{attribute 'GeneratedUsingTerminal: AMP8000-0030-0103-0103'}
{attribute addProperty BoxType "AMP8000-0030-0103-0103"}
{attribute addProperty Id "WcState0AT %I*BOOL1WcState1AT %I*BOOL1InputToggle0AT %I*BOOL1InputToggle1AT %I*BOOL1"}
{attribute addProperty CRC "3038159460"}
{attribute addProperty Size "4"}
TYPE WcState_B516A264 :
STRUCT
	{attribute addProperty Name "WcState0"}
	WcState0 AT %I* : BOOL;
	{attribute addProperty Name "WcState1"}
	WcState1 AT %I* : BOOL;
	{attribute addProperty Name "InputToggle0"}
	InputToggle0 AT %I* : BOOL;
	{attribute addProperty Name "InputToggle1"}
	InputToggle1 AT %I* : BOOL;
END_STRUCT
END_TYPE

(* stored: Version 1.2.0.0, ProductVersion 3.1.4024.9
   DUT WcState_B516A264: Id {10cf3fe7-183a-4c47-ba25-490d12d195a9} *)
